TYPE ST_TaskState :
	STRUCT
		Name	: T_MaxString;
		Busy	: BOOL;
		Error	: BOOL;
		ErrorId : UDINT;
	END_STRUCT
END_TYPE

(* stored: Version 1.1.0.1, ProductVersion 3.1.4026.18
   DUT ST_TaskState: Id {ad6158ba-433c-4120-bd8a-72b9dc1ed2d2} *)
